// Copyright (c) 2024 Loupe (https://loupe.team), provided under the MIT License.
PROGRAM Example
VAR
	myRobotLink : TcAbbLinkin;
	initConfiguration : BOOL := TRUE;
	initConnection : BOOL := TRUE;
	userCommand_GetState : BOOL := TRUE;
	getStateStatus : AbbLinkinRequestStatus_Typ;
	currentState : STRING;
	output : STRING;
END_VAR

// Initialize configuration
IF initConfiguration THEN
	myRobotLink.configuration.rwsIpAddress := '127.0.0.1';
	myRobotLink.configuration.rwsTcpPort := 80;
	myRobotLink.configuration.rwsVersion := ABBLINKIN_RWS_API_VERSION.V2;
	myRobotLink.configuration.rwsUsername := 'Default User';
	myRobotLink.configuration.rwsPassword := 'robotics';
	myRobotLink.configuration.tlsAllowRwsCertSelfSigned := TRUE;
	
	initConfiguration := FALSE;
END_IF

myRobotLink.Cyclic();

/////////////////////////
// Connect
IF initConnection THEN
	myRobotLink.ConnectionStart();
	initConnection := FALSE;
END_IF

/////////////////////////
// Get State

// Send command
IF myRobotLink.readyForCmd AND userCommand_GetState THEN
	myRobotLink.GetRapidState(pStatus := ADR(getStateStatus), pResultState := ADR(currentState));
	userCommand_GetState := FALSE;
END_IF

// Process Results
IF getStateStatus.done THEN
	output := CONCAT('Current state is ', currentState);
ELSIF getStateStatus.error THEN
	output := 'An Error occured.';
END_IF

END_PROGRAM

(* stored: Version 1.1.0.1, ProductVersion 3.1.4024.12
   POU Example: Id {6ae7d968-fc96-4ba1-b6bb-dff0068c2fd8}, SpecialFunc None *)
